FUNCTION_BLOCK FB_Co2FlowModelDeviationHandler
VAR_INPUT
	currentFlow : REAL;
	modeledFlow : REAL;
END_VAR
VAR_OUTPUT
	deviationPercentage : DINT;
END_VAR
VAR
	delta : REAL;
	_maxValue : REAL;
END_VAR


IF currentFlow <> 0 THEN
	delta := modeledFlow - currentFlow;
	
	// Normalize max value to 100 percent
	deviationPercentage := TO_DINT((delta/_maxValue)*100);
	
ELSE
	deviationPercentage := 0;
END_IF

METHOD FB_init : BOOL
VAR_INPUT
	bInitRetains : BOOL; // if TRUE, the retain variables are initialized (warm start / cold start)
	bInCopyCode : BOOL;  // if TRUE, the instance afterwards gets moved into the copy code (online change)
	maxValue : REAL;
END_VAR

_maxValue := maxValue;
END_METHOD

END_FUNCTION_BLOCK

(* stored: Version 1.1.0.1, ProductVersion 3.1.4024.9
   POU FB_Co2FlowModelDeviationHandler: Id {41bdbea2-c2c3-4bcc-af0a-3bfe6b896eda}, SpecialFunc None
   Method FB_init: Id {c9a6c0da-d58b-4075-b4b9-0be02bdcf797} *)
